SUBAPPLICATION Uebung_10c (* SoftKey_F1 auf DigitalOutput_Q1 mit GreenWhiteBackground *)
  (* Standard: 61499-2; Description: Copyright (c) 2023 Meisterschulen am Ostbahnhof This program and the accompanying materials are made available under the terms of the Eclipse Public License 2.0 which is available at https://www.eclipse.org/legal/epl-2.0/ SPDX-License-Identifier: EPL-2.0 *)
  (* Version 1.0, 2023-10-23, Franz Höpfinger, Meisterschulen am Ostbahnhof *)
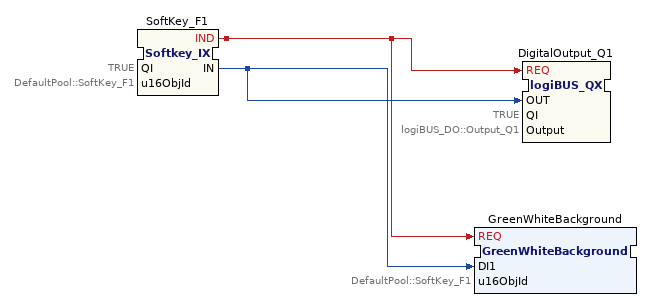
  (* Nachteil: DefaultPool::SoftKey_F1 muss 2x angegeben werden *)
  FBS
    DigitalOutput_Q1 : logiBUS_QX(QI := TRUE, Output := logiBUS_DO::Output_Q1);
    SoftKey_F1 : Softkey_IX(QI := TRUE, u16ObjId := DefaultPool::SoftKey_F1);
  END_FBS
  SUBAPPS
    GreenWhiteBackground : GreenWhiteBackground(u16ObjId := DefaultPool::SoftKey_F1);
  END_SUBAPPS
  EVENT_CONNECTIONS
    SoftKey_F1.IND TO DigitalOutput_Q1.REQ;
    SoftKey_F1.IND TO GreenWhiteBackground.REQ;
  END_CONNECTIONS
  DATA_CONNECTIONS
    SoftKey_F1.IN TO DigitalOutput_Q1.OUT;
    SoftKey_F1.IN TO GreenWhiteBackground.DI1;
  END_CONNECTIONS
END_SUBAPPLICATION
